// TIA Portal V17 export
// export: Created 2022-06-27T13:59:12.3391647Z, ExportSetting WithDefaults, DisplayName Totally Integrated Automation Portal, DisplayVersion V17 Update 3, DisplayName TIA Portal Openness, DisplayVersion V17 Update 3, DisplayName TIA Portal Version Control Interface, DisplayVersion V17, DisplayName SINAMICS Startdrive Advanced, DisplayVersion V17 Update1, DisplayName SINAMICS Startdrive G110M, G120, G120C, G120D, G120P, G115D, DisplayVersion V17 Update1, DisplayName SINAMICS Startdrive G130, G150, S120, S150, SINAMICS MV, S210, DisplayVersion V17 Update1, DisplayName STEP 7 Professional, DisplayVersion V17 Update 3, DisplayName STEP 7 Safety, DisplayVersion V17, DisplayName WinCC UA Professional, DisplayVersion V17 Update 3
FUNCTION_BLOCK "S064_DIGITAL_OUTPUTS"   // FB64, LAD
{ S7_Optimized_Access := 'TRUE' }
VERSION : 0.1
// stored: AutoNumber false, IsIECCheckEnabled false, IsRetainMemResEnabled false, MemoryReserve 100, SetENOAutomatically false, UDAEnableTagReadback false
BEGIN

REGION Network 1: K62-2E - Auxiliary Combustor Fan Drive
END_REGION

REGION Network 2: KM62-3E - Roaster Cyclone Rotary Valve
END_REGION

REGION Network 3: K62-4E - Auxiliary Pump Drive
END_REGION

REGION Network 4: K62-5E - Auxiliary Chamber 1 Drive
END_REGION

REGION Network 5: K62-6E - Auxiliary Chamber 2 Drive
END_REGION

REGION Network 6: KM62-7E - Cooler Cyclone Rotary Valve
END_REGION

REGION Network 7: KM62-8E - Cooler Conveyor Belt
END_REGION

REGION Network 8: KM62-9E - Tilted Screw Conveyor
END_REGION

REGION Network 9: K63-2E - Auxiliary Cooler 1 Drive
END_REGION

REGION Network 10: K63-3E - Auxiliary Cooler 2 Drive
END_REGION

REGION Network 11: KM63-4E - Dryer Cyclone 1 Rotary Valve
END_REGION

REGION Network 12: KM63-5E - Dryer Cyclone 2 Rotary Valve
END_REGION

REGION Network 13: KM63-6E - Cyclones Screw Conveyor
END_REGION

REGION Network 14: K63-7E - Silo 1 Raw Coffee Request
END_REGION

REGION Network 15: K63-8E - Silo 1 Raw Coffee Request
END_REGION

REGION Network 16: K64-2E - Transport Request "catador"
END_REGION

REGION Network 17: K64-3E - Transport Request HVH
END_REGION

REGION Network 18: K64-4E - Combustor Auxiliary Reset
END_REGION

REGION Network 19: K64-5E - Combustor Auxiliary On
END_REGION

REGION Network 20: K64-6E - Combustor Fuel Selection
END_REGION

REGION Network 21: FV78-2E - Chamber 1 Water Plumbing Cleaning
END_REGION

REGION Network 22: FV78-3E - Chamber 2 Water Plumbing Cleaning
END_REGION

REGION Network 23: FV78-4E - Tank Pressurization
END_REGION

REGION Network 24: K92-6E - Chamber 1 Auxiliary Water Pump
END_REGION

REGION Network 25: FV78-6E - Cooler 1 on Fire Emergency
END_REGION

REGION Network 26: K92-7E - Chamber 2 Auxiliary Water Pump
END_REGION

REGION Network 27: FV78-8E - Cooler 2 on Fire Emergency
END_REGION

REGION Network 28: FV78-9E - Silverskin Water Solenoid
END_REGION

REGION Network 29: FV79-2E - Water Tank Relief
END_REGION

REGION Network 30: FV79-3E - Water Tank Intake
END_REGION

REGION Network 31: FV79-4E - Silverskin Emergency Water Solenoid
END_REGION
END_FUNCTION_BLOCK
